FUNCTION_BLOCK reactor
  (* Standard: 61499-2 *)
  (* Version 0.1, 2015-00-13, Th?o, PC_THEO *)
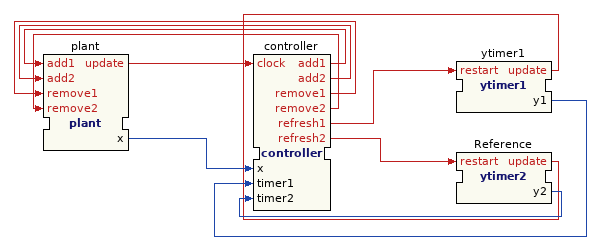
  FBS
    controller : controller;
    plant : plant;
    ytimer1 : ytimer1;
    Reference : ytimer2;
  END_FBS
  EVENT_CONNECTIONS
    controller.add1 TO plant.add1;
    controller.add2 TO plant.add2;
    controller.remove1 TO plant.remove1;
    controller.remove2 TO plant.remove2;
    controller.refresh1 TO ytimer1.restart;
    controller.refresh2 TO Reference.restart;
    plant.update TO controller.clock;
    ytimer1.update TO controller.clock;
    Reference.update TO controller.clock;
  END_CONNECTIONS
  DATA_CONNECTIONS
    plant.x TO controller.x;
    ytimer1.y1 TO controller.timer1;
    Reference.y2 TO controller.timer2;
  END_CONNECTIONS
END_FUNCTION_BLOCK
